{attribute 'qualified_only'}
VAR_GLOBAL
END_VAR

(* stored: Version 1.1.0.1, ProductVersion 3.1.4022.7
   GVL GVL_01_Flag: Id {0acb9164-52a7-4330-9cc9-71148b8b0b93} *)
